# B&R Automation Studio project Foerderband
Automation Studio 4.7.2.98

## Configuration Config1

### Task classes (Cpu.sw)
```
Cyclic#1:
  Program <- Program.prg
Binaries: udbdef, FWRules, TCData, sysconf, Role, User, iomap, ashwd, asiol1, asfw, arconfig, ashwac
Libraries: standard
```

### Hardware
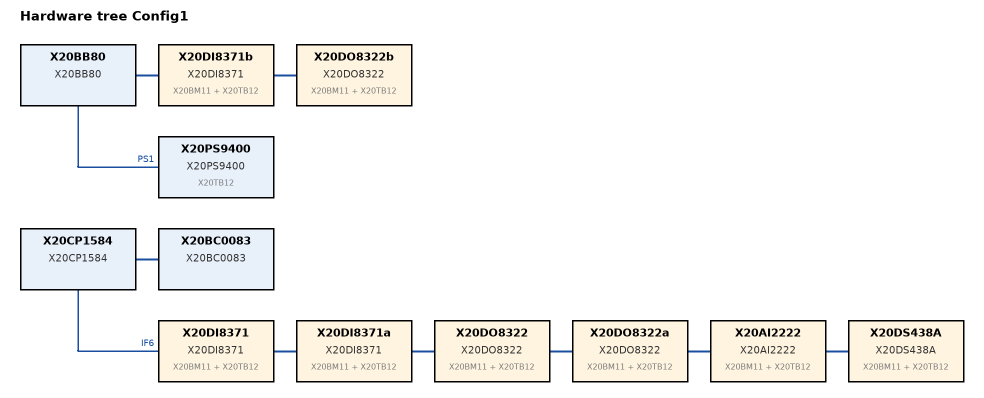
```
X20AI2222 : X20AI2222 v1.0.2.0  [SS1 -> X20TB12d.SS; SL -> X20BM11d.SL1]
X20BB80 : X20BB80 v1.0.2.0
X20BC0083 : X20BC0083 v2.9.0.0  [PLK1 -> X20CP1584.IF3 [Cable Type=PowerlinkCable, Length=10, Version=1.0.0.2]; SL -> X20BB80.SL1]
X20BM11 : X20BM11 v1.0.0.1  [X2X1 -> X20CP1584.IF6]
X20BM11a : X20BM11 v1.0.0.1  [X2X1 -> X20BM11.X2X2]
X20BM11b : X20BM11 v1.0.0.1  [X2X1 -> X20BM11a.X2X2]
X20BM11c : X20BM11 v1.0.0.1  [X2X1 -> X20BM11b.X2X2]
X20BM11d : X20BM11 v1.0.0.1  [X2X1 -> X20BM11c.X2X2]
X20BM11e : X20BM11 v1.0.0.1  [X2X1 -> X20BM11d.X2X2]
X20BM11f : X20BM11 v1.0.0.1  [X2X1 -> X20BB80.IF1]
X20BM11h : X20BM11 v1.0.0.1  [X2X1 -> X20BM11f.X2X2]
X20CP1584 : X20CP1584 v1.6.0.0
  Connector IF2:
    ActivateDevice = 1
    Mode = Manual
    InternetAddress = 10.36.37.4
    SubnetMask = 255.255.255.0
  ConfigurationID = Foerderband_Config1
X20DI8371 : X20DI8371 v1.0.2.0  [SS1 -> X20TB12.SS; SL -> X20BM11.SL1]
X20DI8371a : X20DI8371 v1.0.2.0  [SS1 -> X20TB12a.SS; SL -> X20BM11a.SL1]
X20DI8371b : X20DI8371 v1.0.2.0  [SS1 -> X20TB12f.SS; SL -> X20BM11f.SL1]
X20DO8322 : X20DO8322 v1.1.0.0  [SS1 -> X20TB12b.SS; SL -> X20BM11b.SL1]
X20DO8322a : X20DO8322 v1.1.0.0  [SS1 -> X20TB12c.SS; SL -> X20BM11c.SL1]
X20DO8322b : X20DO8322 v1.1.0.0  [SS1 -> X20TB12i.SS; SL -> X20BM11h.SL1]
X20DS438A : X20DS438A v1.9.1.0  [SS1 -> X20TB12e.SS; SL -> X20BM11e.SL1]
  DtmRef = FBD.BRIOLinkModuleDTM.DTMCore.X20DS438A
  DtmId = 94a64cda-18e3-4e02-9df8-4711ba989a67
  CommDtmId = c69bdead-edba-4600-ad5b-e2199e73abc9
  RequiresDTMBuild = true
  ConfigFile = Communication.dtm
  ConfigModule = asiol1
X20PS9400 : X20PS9400 v1.0.2.4  [SS1 -> X20TB12g.SS; PS -> X20BB80.PS1]
X20TB12 : X20TB12 v1.0.0.0
X20TB12a : X20TB12 v1.0.0.0
X20TB12b : X20TB12 v1.0.0.0
X20TB12c : X20TB12 v1.0.0.0
X20TB12d : X20TB12 v1.0.0.0
X20TB12e : X20TB12 v1.0.0.0
X20TB12f : X20TB12 v1.0.0.0
X20TB12g : X20TB12 v1.0.0.0
X20TB12i : X20TB12 v1.0.0.0
```

### IoMap.iom - X20CP1584/IoMap.iom
```iecst
VAR_CONFIG
	DI_Band_links AT %IX."X20DI8371".DigitalInput01;
	DI_Band_rechts AT %IX."X20DI8371".DigitalInput02;
	DI_Koppel_rechts AT %IX."X20DI8371".DigitalInput03;
	DI_Koppel_links AT %IX."X20DI8371".DigitalInput04;
	DI_Stopper AT %IX."X20DI8371".DigitalInput05;
	DI_NOTAUS AT %IX."X20DI8371".DigitalInput06;
	DI_Drehgeber_1 AT %IX."X20DI8371".DigitalInput07;
	DI_Drehgeber_2  AT %IX."X20DI8371".DigitalInput08;
	DI_Start AT %IX."X20DI8371a".DigitalInput01;
	DI_Stop AT %IX."X20DI8371a".DigitalInput02;
	DI_RESET AT %IX."X20DI8371a".DigitalInput03;
	DI_Wahl AT %IX."X20DI8371a".DigitalInput04;
	DO_Antrieb_rechts AT %QX."X20DO8322".DigitalOutput01;
	DO_Antrieb_links AT %QX."X20DO8322".DigitalOutput02;
	DO_schleichgang AT %QX."X20DO8322".DigitalOutput03;
	DO_Stopper AT %QX."X20DO8322".DigitalOutput04;
	DO_Koppel_links AT %QX."X20DO8322".DigitalOutput05;
	DO_Koppel_rechts AT %QX."X20DO8322".DigitalOutput06;
	DO_gruen AT %QX."X20DO8322a".DigitalOutput01;
	DO_weiss AT %QX."X20DO8322a".DigitalOutput02;
	DO_Q1 AT %QX."X20DO8322a".DigitalOutput03;
	DO_Q2 AT %QX."X20DO8322a".DigitalOutput04;
	AI_Potentiometer_1 AT %IW."X20AI2222".AnalogInput01;
	AI_Potentiometer_2 AT %IW."X20AI2222".AnalogInput02;
END_VAR
```

## Configuration station_1

### Task classes (Cpu.sw)
```
Cyclic#1:
  Foerderban <- Foerderband.prg
  stat_1 <- stat_1.prg
  Foerdeband <- FoerdebandWatch.prg
Binaries: udbdef, FWRules, TCData, sysconf, Role, User, iomap, ashwd, asiol1, asfw, arconfig, ashwac
Libraries: standard
```

### Hardware
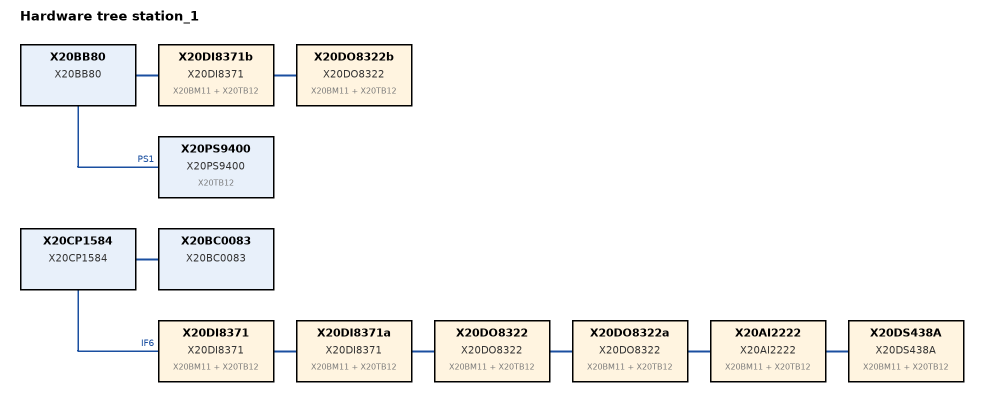
```
X20AI2222 : X20AI2222 v1.0.2.0  [SS1 -> X20TB12d.SS; SL -> X20BM11d.SL1]
X20BB80 : X20BB80 v1.0.2.0
X20BC0083 : X20BC0083 v2.9.0.0  [PLK1 -> X20CP1584.IF3 [Cable Type=PowerlinkCable, Length=10, Version=1.0.0.2]; SL -> X20BB80.SL1]
X20BM11 : X20BM11 v1.0.0.1  [X2X1 -> X20CP1584.IF6]
X20BM11a : X20BM11 v1.0.0.1  [X2X1 -> X20BM11.X2X2]
X20BM11b : X20BM11 v1.0.0.1  [X2X1 -> X20BM11a.X2X2]
X20BM11c : X20BM11 v1.0.0.1  [X2X1 -> X20BM11b.X2X2]
X20BM11d : X20BM11 v1.0.0.1  [X2X1 -> X20BM11c.X2X2]
X20BM11e : X20BM11 v1.0.0.1  [X2X1 -> X20BM11d.X2X2]
X20BM11f : X20BM11 v1.0.0.1  [X2X1 -> X20BB80.IF1]
X20BM11h : X20BM11 v1.0.0.1  [X2X1 -> X20BM11f.X2X2]
X20CP1584 : X20CP1584 v1.6.0.0
  Connector IF2:
    ActivateDevice = 1
    Mode = Manual
    InternetAddress = 10.36.37.1
    SubnetMask = 255.255.255.0
  ConfigurationID = Foerderband_Config1
X20DI8371 : X20DI8371 v1.0.2.0  [SS1 -> X20TB12.SS; SL -> X20BM11.SL1]
X20DI8371a : X20DI8371 v1.0.2.0  [SS1 -> X20TB12a.SS; SL -> X20BM11a.SL1]
X20DI8371b : X20DI8371 v1.0.2.0  [SS1 -> X20TB12f.SS; SL -> X20BM11f.SL1]
X20DO8322 : X20DO8322 v1.1.0.0  [SS1 -> X20TB12b.SS; SL -> X20BM11b.SL1]
X20DO8322a : X20DO8322 v1.1.0.0  [SS1 -> X20TB12c.SS; SL -> X20BM11c.SL1]
X20DO8322b : X20DO8322 v1.1.0.0  [SS1 -> X20TB12i.SS; SL -> X20BM11h.SL1]
X20DS438A : X20DS438A v1.9.1.0  [SS1 -> X20TB12e.SS; SL -> X20BM11e.SL1]
  DtmRef = FBD.BRIOLinkModuleDTM.DTMCore.X20DS438A
  DtmId = 94a64cda-18e3-4e02-9df8-4711ba989a67
  CommDtmId = c69bdead-edba-4600-ad5b-e2199e73abc9
  RequiresDTMBuild = true
  ConfigFile = Communication.dtm
  ConfigModule = asiol1
X20PS9400 : X20PS9400 v1.0.2.4  [SS1 -> X20TB12g.SS; PS -> X20BB80.PS1]
X20TB12 : X20TB12 v1.0.0.0
X20TB12a : X20TB12 v1.0.0.0
X20TB12b : X20TB12 v1.0.0.0
X20TB12c : X20TB12 v1.0.0.0
X20TB12d : X20TB12 v1.0.0.0
X20TB12e : X20TB12 v1.0.0.0
X20TB12f : X20TB12 v1.0.0.0
X20TB12g : X20TB12 v1.0.0.0
X20TB12i : X20TB12 v1.0.0.0
```

### IoMap.iom - X20CP1584/IoMap.iom
```iecst
VAR_CONFIG
	DI_Band_links AT %IX."X20DI8371".DigitalInput01;
	DI_Band_rechts AT %IX."X20DI8371".DigitalInput02;
	DI_Koppel_rechts AT %IX."X20DI8371".DigitalInput03;
	DI_Koppel_links AT %IX."X20DI8371".DigitalInput04;
	DI_Stopper AT %IX."X20DI8371".DigitalInput05;
	DI_NOTAUS AT %IX."X20DI8371".DigitalInput06;
	DI_Drehgeber_1 AT %IX."X20DI8371".DigitalInput07;
	DI_Drehgeber_2 AT %IX."X20DI8371".DigitalInput08;
	DI_Start AT %IX."X20DI8371a".DigitalInput01;
	DI_Stop AT %IX."X20DI8371a".DigitalInput02;
	DI_RESET AT %IX."X20DI8371a".DigitalInput03;
	DI_Wahl AT %IX."X20DI8371a".DigitalInput04;
	DO_Antrieb_rechts AT %QX."X20DO8322".DigitalOutput01;
	DO_Antrieb_links AT %QX."X20DO8322".DigitalOutput02;
	DO_schleichgang AT %QX."X20DO8322".DigitalOutput03;
	DO_Stopper AT %QX."X20DO8322".DigitalOutput04;
	DO_Koppel_links AT %QX."X20DO8322".DigitalOutput05;
	DO_Koppel_rechts AT %QX."X20DO8322".DigitalOutput06;
	DO_gruen AT %QX."X20DO8322a".DigitalOutput01;
	DO_weiss AT %QX."X20DO8322a".DigitalOutput02;
	DO_Q1 AT %QX."X20DO8322a".DigitalOutput03;
	DO_Q2 AT %QX."X20DO8322a".DigitalOutput04;
	AI_Potentiometer_1 AT %IW."X20AI2222".AnalogInput01;
	AI_Potentiometer_2 AT %IW."X20AI2222".AnalogInput02;
	::DI_Ident_1 AT %IX."X20DI8371a".DigitalInput05;
	::DI_Ident_2 AT %IX."X20DI8371a".DigitalInput06;
	::DI_Ident_3 AT %IX."X20DI8371a".DigitalInput07;
	::DI_Ident_4 AT %IX."X20DI8371a".DigitalInput08;
	DI_X_axis_links  AT %IX."X20DI8371b".DigitalInput01;
	DI_X_axis_recht AT %IX."X20DI8371b".DigitalInput02;
	DI_Frontschale_korr  AT %IX."X20DI8371b".DigitalInput03;
	DI_Frontschale_vorh  AT %IX."X20DI8371b".DigitalInput04;
	DI_Z_axis_oben  AT %IX."X20DI8371b".DigitalInput05;
	DI_Z_axis_unten  AT %IX."X20DI8371b".DigitalInput06;
	DI_Deckel_bereits_vorh  AT %IX."X20DI8371b".DigitalInput07;
	DO_X_axis_nach_links  AT %QX."X20DO8322b".DigitalOutput01;
	DO_X_axis_nach_rechts AT %QX."X20DO8322b".DigitalOutput02;
	DO_Z_axis_nach_oben  AT %QX."X20DO8322b".DigitalOutput03;
	DO_Z_axis_nach_unten  AT %QX."X20DO8322b".DigitalOutput04;
	DO_Z_axis_Klemmung  AT %QX."X20DO8322b".DigitalOutput05;
	DO_Bohrer1  AT %QX."X20DO8322b".DigitalOutput06;
	DO_Bohrer2  AT %QX."X20DO8322b".DigitalOutput07;
END_VAR
```

## Configuration station_2

### Task classes (Cpu.sw)
```
Cyclic#1:
  stat_2 <- stat_2.prg
  Foerderban <- Foerderband.prg
  Program <- (binary)
Binaries: udbdef, FWRules, TCData, sysconf, Role, User, iomap, ashwd, asiol1, asfw, arconfig, ashwac
Libraries: standard
```

### Hardware
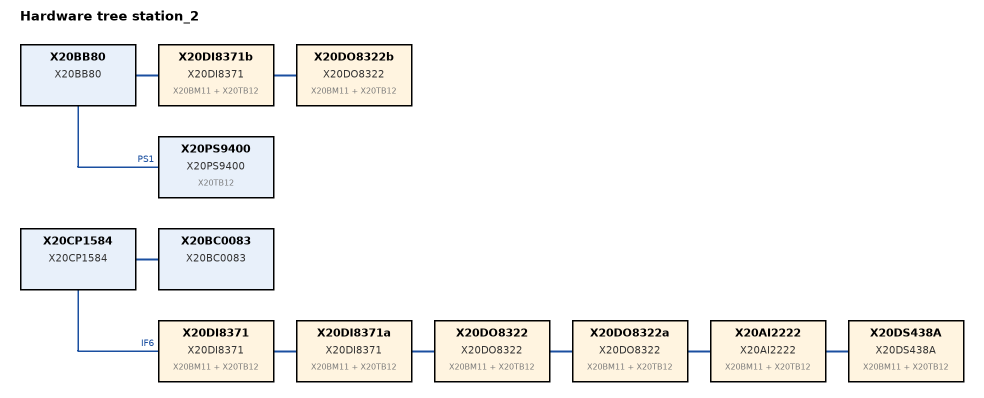
```
X20AI2222 : X20AI2222 v1.0.2.0  [SS1 -> X20TB12d.SS; SL -> X20BM11d.SL1]
X20BB80 : X20BB80 v1.0.2.0
X20BC0083 : X20BC0083 v2.9.0.0  [PLK1 -> X20CP1584.IF3 [Cable Type=PowerlinkCable, Length=10, Version=1.0.0.2]; SL -> X20BB80.SL1]
X20BM11 : X20BM11 v1.0.0.1  [X2X1 -> X20CP1584.IF6]
X20BM11a : X20BM11 v1.0.0.1  [X2X1 -> X20BM11.X2X2]
X20BM11b : X20BM11 v1.0.0.1  [X2X1 -> X20BM11a.X2X2]
X20BM11c : X20BM11 v1.0.0.1  [X2X1 -> X20BM11b.X2X2]
X20BM11d : X20BM11 v1.0.0.1  [X2X1 -> X20BM11c.X2X2]
X20BM11e : X20BM11 v1.0.0.1  [X2X1 -> X20BM11d.X2X2]
X20BM11f : X20BM11 v1.0.0.1  [X2X1 -> X20BB80.IF1]
X20BM11h : X20BM11 v1.0.0.1  [X2X1 -> X20BM11f.X2X2]
X20CP1584 : X20CP1584 v1.6.0.0
  Connector IF2:
    ActivateDevice = 1
    Mode = Manual
    InternetAddress = 10.36.37.2
    SubnetMask = 255.255.255.0
  ConfigurationID = Foerderband_Config1
X20DI8371 : X20DI8371 v1.0.2.0  [SS1 -> X20TB12.SS; SL -> X20BM11.SL1]
X20DI8371a : X20DI8371 v1.0.2.0  [SS1 -> X20TB12a.SS; SL -> X20BM11a.SL1]
X20DI8371b : X20DI8371 v1.0.2.0  [SS1 -> X20TB12f.SS; SL -> X20BM11f.SL1]
X20DO8322 : X20DO8322 v1.1.0.0  [SS1 -> X20TB12b.SS; SL -> X20BM11b.SL1]
X20DO8322a : X20DO8322 v1.1.0.0  [SS1 -> X20TB12c.SS; SL -> X20BM11c.SL1]
X20DO8322b : X20DO8322 v1.1.0.0  [SS1 -> X20TB12i.SS; SL -> X20BM11h.SL1]
X20DS438A : X20DS438A v1.9.1.0  [SS1 -> X20TB12e.SS; SL -> X20BM11e.SL1]
  DtmRef = FBD.BRIOLinkModuleDTM.DTMCore.X20DS438A
  DtmId = 94a64cda-18e3-4e02-9df8-4711ba989a67
  CommDtmId = c69bdead-edba-4600-ad5b-e2199e73abc9
  RequiresDTMBuild = true
  ConfigFile = Communication.dtm
  ConfigModule = asiol1
X20PS9400 : X20PS9400 v1.0.2.4  [SS1 -> X20TB12g.SS; PS -> X20BB80.PS1]
X20TB12 : X20TB12 v1.0.0.0
X20TB12a : X20TB12 v1.0.0.0
X20TB12b : X20TB12 v1.0.0.0
X20TB12c : X20TB12 v1.0.0.0
X20TB12d : X20TB12 v1.0.0.0
X20TB12e : X20TB12 v1.0.0.0
X20TB12f : X20TB12 v1.0.0.0
X20TB12g : X20TB12 v1.0.0.0
X20TB12i : X20TB12 v1.0.0.0
```

### IoMap.iom - X20CP1584/IoMap.iom
```iecst
VAR_CONFIG
	DI_Band_links AT %IX."X20DI8371".DigitalInput01;
	DI_Band_rechts AT %IX."X20DI8371".DigitalInput02;
	DI_Koppel_rechts AT %IX."X20DI8371".DigitalInput03;
	DI_Koppel_links AT %IX."X20DI8371".DigitalInput04;
	DI_Stopper AT %IX."X20DI8371".DigitalInput05;
	DI_NOTAUS AT %IX."X20DI8371".DigitalInput06;
	DI_Drehgeber_1 AT %IX."X20DI8371".DigitalInput07;
	DI_Drehgeber_2 AT %IX."X20DI8371".DigitalInput08;
	DI_Start AT %IX."X20DI8371a".DigitalInput01;
	DI_Stop AT %IX."X20DI8371a".DigitalInput02;
	DI_RESET AT %IX."X20DI8371a".DigitalInput03;
	DI_Wahl AT %IX."X20DI8371a".DigitalInput04;
	DO_Antrieb_rechts AT %QX."X20DO8322".DigitalOutput01;
	DO_Antrieb_links AT %QX."X20DO8322".DigitalOutput02;
	DO_schleichgang AT %QX."X20DO8322".DigitalOutput03;
	DO_Stopper AT %QX."X20DO8322".DigitalOutput04;
	DO_Koppel_links AT %QX."X20DO8322".DigitalOutput05;
	DO_Koppel_rechts AT %QX."X20DO8322".DigitalOutput06;
	DO_gruen AT %QX."X20DO8322a".DigitalOutput01;
	DO_weiss AT %QX."X20DO8322a".DigitalOutput02;
	DO_Q1 AT %QX."X20DO8322a".DigitalOutput03;
	DO_Q2 AT %QX."X20DO8322a".DigitalOutput04;
	AI_Potentiometer_1 AT %IW."X20AI2222".AnalogInput01;
	AI_Potentiometer_2 AT %IW."X20AI2222".AnalogInput02;
	::DI_Ident_1 AT %IX."X20DI8371a".DigitalInput05;
	::DI_Ident_2 AT %IX."X20DI8371a".DigitalInput06;
	::DI_Ident_3 AT %IX."X20DI8371a".DigitalInput07;
	::DI_Ident_4 AT %IX."X20DI8371a".DigitalInput08;
	DI_Hubzylinder_oben  AT %IX."X20DI8371b".DigitalInput01;
	DI_Hubzylinder_unten  AT %IX."X20DI8371b".DigitalInput02;
	DI_untere_Klinge  AT %IX."X20DI8371b".DigitalInput03;
	DI_obere_Klinge  AT %IX."X20DI8371b".DigitalInput04;
	DI_Mag_leer  AT %IX."X20DI8371b".DigitalInput05;
	DI_Palette  AT %IX."X20DI8371b".DigitalInput06;
	DI_Frontschale  AT %IX."X20DI8371b".DigitalInput07;
	DO_Hubzylinder_auf  AT %QX."X20DO8322b".DigitalOutput01;
	DO_Hubzylinder_ab  AT %QX."X20DO8322b".DigitalOutput02;
	DO_Vereinzler_close  AT %QX."X20DO8322b".DigitalOutput03;
	DO_Vereinzler_open  AT %QX."X20DO8322b".DigitalOutput04;
	DO_Zylinderklemmung  AT %QX."X20DO8322b".DigitalOutput05;
END_VAR
```

## Configuration station_3

### Hardware
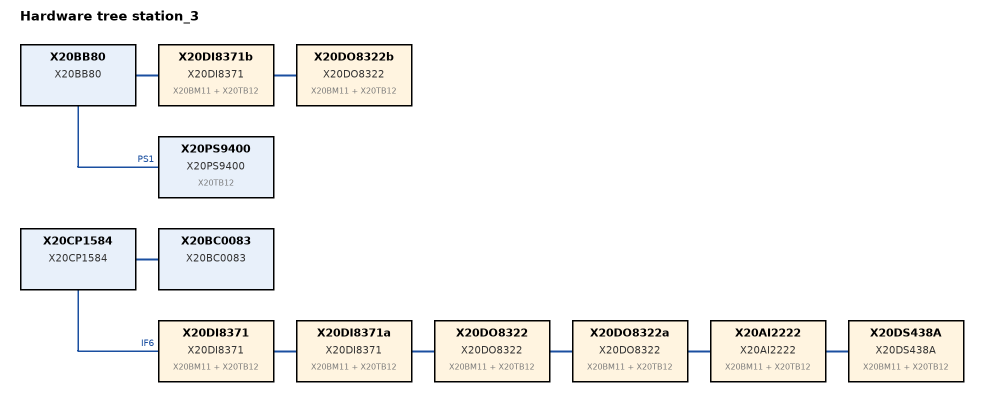
```
X20AI2222 : X20AI2222 v1.0.2.0  [SS1 -> X20TB12d.SS; SL -> X20BM11d.SL1]
X20BB80 : X20BB80 v1.0.2.0
X20BC0083 : X20BC0083 v2.9.0.0  [PLK1 -> X20CP1584.IF3 [Cable Type=PowerlinkCable, Length=10, Version=1.0.0.2]; SL -> X20BB80.SL1]
X20BM11 : X20BM11 v1.0.0.1  [X2X1 -> X20CP1584.IF6]
X20BM11a : X20BM11 v1.0.0.1  [X2X1 -> X20BM11.X2X2]
X20BM11b : X20BM11 v1.0.0.1  [X2X1 -> X20BM11a.X2X2]
X20BM11c : X20BM11 v1.0.0.1  [X2X1 -> X20BM11b.X2X2]
X20BM11d : X20BM11 v1.0.0.1  [X2X1 -> X20BM11c.X2X2]
X20BM11e : X20BM11 v1.0.0.1  [X2X1 -> X20BM11d.X2X2]
X20BM11f : X20BM11 v1.0.0.1  [X2X1 -> X20BB80.IF1]
X20BM11h : X20BM11 v1.0.0.1  [X2X1 -> X20BM11f.X2X2]
X20CP1584 : X20CP1584 v1.6.0.0
  Connector IF2:
    ActivateDevice = 1
    Mode = Manual
    InternetAddress = 10.36.37.3
    SubnetMask = 255.255.255.0
  ConfigurationID = Foerderband_Config1
X20DI8371 : X20DI8371 v1.0.2.0  [SS1 -> X20TB12.SS; SL -> X20BM11.SL1]
X20DI8371a : X20DI8371 v1.0.2.0  [SS1 -> X20TB12a.SS; SL -> X20BM11a.SL1]
X20DI8371b : X20DI8371 v1.0.2.0  [SS1 -> X20TB12f.SS; SL -> X20BM11f.SL1]
X20DO8322 : X20DO8322 v1.1.0.0  [SS1 -> X20TB12b.SS; SL -> X20BM11b.SL1]
X20DO8322a : X20DO8322 v1.1.0.0  [SS1 -> X20TB12c.SS; SL -> X20BM11c.SL1]
X20DO8322b : X20DO8322 v1.1.0.0  [SS1 -> X20TB12i.SS; SL -> X20BM11h.SL1]
X20DS438A : X20DS438A v1.9.1.0  [SS1 -> X20TB12e.SS; SL -> X20BM11e.SL1]
  DtmRef = FBD.BRIOLinkModuleDTM.DTMCore.X20DS438A
  DtmId = 94a64cda-18e3-4e02-9df8-4711ba989a67
  CommDtmId = c69bdead-edba-4600-ad5b-e2199e73abc9
  RequiresDTMBuild = true
  ConfigFile = Communication.dtm
  ConfigModule = asiol1
X20PS9400 : X20PS9400 v1.0.2.4  [SS1 -> X20TB12g.SS; PS -> X20BB80.PS1]
X20TB12 : X20TB12 v1.0.0.0
X20TB12a : X20TB12 v1.0.0.0
X20TB12b : X20TB12 v1.0.0.0
X20TB12c : X20TB12 v1.0.0.0
X20TB12d : X20TB12 v1.0.0.0
X20TB12e : X20TB12 v1.0.0.0
X20TB12f : X20TB12 v1.0.0.0
X20TB12g : X20TB12 v1.0.0.0
X20TB12i : X20TB12 v1.0.0.0
```

### IoMap.iom - X20CP1584/IoMap.iom
```iecst
VAR_CONFIG
	DI_Band_links AT %IX."X20DI8371".DigitalInput01;
	DI_Band_rechts AT %IX."X20DI8371".DigitalInput02;
	DI_Koppel_rechts AT %IX."X20DI8371".DigitalInput03;
	DI_Koppel_links AT %IX."X20DI8371".DigitalInput04;
	DI_Stopper AT %IX."X20DI8371".DigitalInput05;
	DI_NOTAUS AT %IX."X20DI8371".DigitalInput06;
	DI_Drehgeber_1 AT %IX."X20DI8371".DigitalInput07;
	DI_Drehgeber_2 AT %IX."X20DI8371".DigitalInput08;
	DI_Start AT %IX."X20DI8371a".DigitalInput01;
	DI_Stop AT %IX."X20DI8371a".DigitalInput02;
	DI_RESET AT %IX."X20DI8371a".DigitalInput03;
	DI_Wahl AT %IX."X20DI8371a".DigitalInput04;
	DO_Antrieb_rechts AT %QX."X20DO8322".DigitalOutput01;
	DO_Antrieb_links AT %QX."X20DO8322".DigitalOutput02;
	DO_schleichgang AT %QX."X20DO8322".DigitalOutput03;
	DO_Stopper AT %QX."X20DO8322".DigitalOutput04;
	DO_Koppel_links AT %QX."X20DO8322".DigitalOutput05;
	DO_Koppel_rechts AT %QX."X20DO8322".DigitalOutput06;
	DO_gruen AT %QX."X20DO8322a".DigitalOutput01;
	DO_weiss AT %QX."X20DO8322a".DigitalOutput02;
	DO_Q1 AT %QX."X20DO8322a".DigitalOutput03;
	DO_Q2 AT %QX."X20DO8322a".DigitalOutput04;
	AI_Potentiometer_1 AT %IW."X20AI2222".AnalogInput01;
	AI_Potentiometer_2 AT %IW."X20AI2222".AnalogInput02;
	::DI_Ident_1 AT %IX."X20DI8371a".DigitalInput05;
	::DI_Ident_2 AT %IX."X20DI8371a".DigitalInput06;
	::DI_Ident_3 AT %IX."X20DI8371a".DigitalInput07;
	::DI_Ident_4 AT %IX."X20DI8371a".DigitalInput08;
	DI_Hubzylinder_oben_stat3 AT %IX."X20DI8371b".DigitalInput01;
	DI_Hubzylinder_unten_stat3 AT %IX."X20DI8371b".DigitalInput02;
	DI_Frontschale_vorhanden AT %IX."X20DI8371b".DigitalInput03;
	DO_Hubzylinder_auf_stat3 AT %QX."X20DO8322b".DigitalOutput01;
	DO_Hubzylinder_ab_stat3 AT %QX."X20DO8322b".DigitalOutput02;
END_VAR
```

## Configuration station_4

### Task classes (Cpu.sw)
```
Cyclic#1:
  Foerderban <- Foerderband.prg
  stat_4 <- stat_4.prg
Binaries: udbdef, FWRules, TCData, sysconf, Role, User, iomap, ashwd, asiol1, asfw, arconfig, ashwac
Libraries: standard
```

### IoMap.iom - X20CP1584/IoMap.iom
```iecst
VAR_CONFIG
	DI_Band_links AT %IX."X20DI8371".DigitalInput01;
	DI_Band_rechts AT %IX."X20DI8371".DigitalInput02;
	DI_Koppel_rechts AT %IX."X20DI8371".DigitalInput03;
	DI_Koppel_links AT %IX."X20DI8371".DigitalInput04;
	DI_Stopper AT %IX."X20DI8371".DigitalInput05;
	DI_NOTAUS AT %IX."X20DI8371".DigitalInput06;
	DI_Drehgeber_1 AT %IX."X20DI8371".DigitalInput07;
	DI_Drehgeber_2 AT %IX."X20DI8371".DigitalInput08;
	DI_Start AT %IX."X20DI8371a".DigitalInput01;
	DI_Stop AT %IX."X20DI8371a".DigitalInput02;
	DI_RESET AT %IX."X20DI8371a".DigitalInput03;
	DI_Wahl AT %IX."X20DI8371a".DigitalInput04;
	DO_Antrieb_rechts AT %QX."X20DO8322".DigitalOutput01;
	DO_Antrieb_links AT %QX."X20DO8322".DigitalOutput02;
	DO_schleichgang AT %QX."X20DO8322".DigitalOutput03;
	DO_Stopper AT %QX."X20DO8322".DigitalOutput04;
	DO_Koppel_links AT %QX."X20DO8322".DigitalOutput05;
	DO_Koppel_rechts AT %QX."X20DO8322".DigitalOutput06;
	DO_gruen AT %QX."X20DO8322a".DigitalOutput01;
	DO_weiss AT %QX."X20DO8322a".DigitalOutput02;
	DO_Q1 AT %QX."X20DO8322a".DigitalOutput03;
	DO_Q2 AT %QX."X20DO8322a".DigitalOutput04;
	AI_Potentiometer_1 AT %IW."X20AI2222".AnalogInput01;
	AI_Potentiometer_2 AT %IW."X20AI2222".AnalogInput02;
	::DI_Ident_1 AT %IX."X20DI8371a".DigitalInput05;
	::DI_Ident_2 AT %IX."X20DI8371a".DigitalInput06;
	::DI_Ident_3 AT %IX."X20DI8371a".DigitalInput07;
	::DI_Ident_4 AT %IX."X20DI8371a".DigitalInput08;
	DI_Hubzylinder_oben AT %IX."X20DI8371b".DigitalInput01;
	DI_Hubzylinder_unten AT %IX."X20DI8371b".DigitalInput02;
	DI_phi_0 AT %IX."X20DI8371b".DigitalInput03;
	DI_phi_180 AT %IX."X20DI8371b".DigitalInput04;
	DI_Greifer_open AT %IX."X20DI8371b".DigitalInput05;
	DI_Greifer_closed AT %IX."X20DI8371b".DigitalInput06;
	DI_Stau AT %IX."X20DI8371b".DigitalInput07;
	DI_Frontschale AT %IX."X20DI8371b".DigitalInput08;
	DO_Hubzylinder_auf AT %QX."X20DO8322b".DigitalOutput01;
	DO_Hubzylinder_ab AT %QX."X20DO8322b".DigitalOutput02;
	DO_phi_0 AT %QX."X20DO8322b".DigitalOutput03;
	DO_phi_180 AT %QX."X20DO8322b".DigitalOutput04;
	DO_Greifer_open AT %QX."X20DO8322b".DigitalOutput05;
	DO_Greifer_close AT %QX."X20DO8322b".DigitalOutput06;
	DO_Zylinderklemmung AT %QX."X20DO8322b".DigitalOutput07;
END_VAR
```

## Configuration station_5

CPU X20CP1584, AutomationRuntime A4.73, Build 4.1.2, Vc V4.72.0

### Task classes (Cpu.sw)
```
Cyclic#1:
  Foerderban <- Foerderband.prg
  Program <- (binary)
  stat_5 <- stat_5.prg
Binaries: udbdef, FWRules, TCData, sysconf, Role, User, iomap, ashwd, asiol1, asfw, arconfig, ashwac
Libraries: standard
```

### Hardware
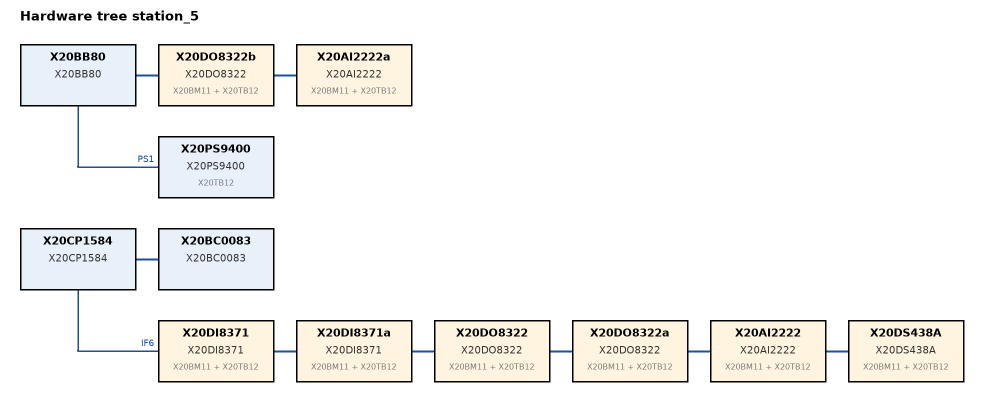
```
X20AI2222 : X20AI2222 v1.0.2.0  [SS1 -> X20TB12d.SS; SL -> X20BM11d.SL1]
X20AI2222a : X20AI2222 v1.0.2.0  [SS1 -> X20TB12h.SS; SL -> X20BM11g.SL1]
X20BB80 : X20BB80 v1.0.2.0
X20BC0083 : X20BC0083 v2.9.0.0  [PLK1 -> X20CP1584.IF3 [Cable Type=PowerlinkCable, Length=10, Version=1.0.0.2]; SL -> X20BB80.SL1]
X20BM11 : X20BM11 v1.0.0.1  [X2X1 -> X20CP1584.IF6]
X20BM11a : X20BM11 v1.0.0.1  [X2X1 -> X20BM11.X2X2]
X20BM11b : X20BM11 v1.0.0.1  [X2X1 -> X20BM11a.X2X2]
X20BM11c : X20BM11 v1.0.0.1  [X2X1 -> X20BM11b.X2X2]
X20BM11d : X20BM11 v1.0.0.1  [X2X1 -> X20BM11c.X2X2]
X20BM11e : X20BM11 v1.0.0.1  [X2X1 -> X20BM11d.X2X2]
X20BM11f : X20BM11 v1.0.0.1  [X2X1 -> X20BB80.IF1]
X20BM11g : X20BM11 v1.0.0.1  [X2X1 -> X20BM11f.X2X2]
X20CP1584 : X20CP1584 v1.6.0.0
  Connector IF2:
    ActivateDevice = 1
    Mode = Manual
    InternetAddress = 10.36.37.5
    SubnetMask = 255.255.255.0
  ConfigurationID = Foerderband_Config1
X20DI8371 : X20DI8371 v1.0.2.0  [SS1 -> X20TB12.SS; SL -> X20BM11.SL1]
X20DI8371a : X20DI8371 v1.0.2.0  [SS1 -> X20TB12a.SS; SL -> X20BM11a.SL1]
X20DO8322 : X20DO8322 v1.1.0.0  [SS1 -> X20TB12b.SS; SL -> X20BM11b.SL1]
X20DO8322a : X20DO8322 v1.1.0.0  [SS1 -> X20TB12c.SS; SL -> X20BM11c.SL1]
X20DO8322b : X20DO8322 v1.1.0.0  [SS1 -> X20TB12f.SS; SL -> X20BM11f.SL1]
X20DS438A : X20DS438A v1.9.1.0  [SS1 -> X20TB12e.SS; SL -> X20BM11e.SL1]
  DtmRef = FBD.BRIOLinkModuleDTM.DTMCore.X20DS438A
  DtmId = 94a64cda-18e3-4e02-9df8-4711ba989a67
  CommDtmId = c69bdead-edba-4600-ad5b-e2199e73abc9
  RequiresDTMBuild = true
  ConfigFile = Communication.dtm
  ConfigModule = asiol1
X20PS9400 : X20PS9400 v1.0.2.4  [SS1 -> X20TB12g.SS; PS -> X20BB80.PS1]
X20TB12 : X20TB12 v1.0.0.0
X20TB12a : X20TB12 v1.0.0.0
X20TB12b : X20TB12 v1.0.0.0
X20TB12c : X20TB12 v1.0.0.0
X20TB12d : X20TB12 v1.0.0.0
X20TB12e : X20TB12 v1.0.0.0
X20TB12f : X20TB12 v1.0.0.0
X20TB12g : X20TB12 v1.0.0.0
X20TB12h : X20TB12 v1.0.0.0
```

### IoMap.iom - X20CP1584/IoMap.iom
```iecst
VAR_CONFIG
	DI_Band_links AT %IX."X20DI8371".DigitalInput01;
	DI_Band_rechts AT %IX."X20DI8371".DigitalInput02;
	DI_Koppel_rechts AT %IX."X20DI8371".DigitalInput03;
	DI_Koppel_links AT %IX."X20DI8371".DigitalInput04;
	DI_Stopper AT %IX."X20DI8371".DigitalInput05;
	DI_NOTAUS AT %IX."X20DI8371".DigitalInput06;
	DI_Drehgeber_1 AT %IX."X20DI8371".DigitalInput07;
	DI_Drehgeber_2 AT %IX."X20DI8371".DigitalInput08;
	DI_Start AT %IX."X20DI8371a".DigitalInput01;
	DI_Stop AT %IX."X20DI8371a".DigitalInput02;
	DI_RESET AT %IX."X20DI8371a".DigitalInput03;
	DI_Wahl AT %IX."X20DI8371a".DigitalInput04;
	DO_Antrieb_rechts AT %QX."X20DO8322".DigitalOutput01;
	DO_Antrieb_links AT %QX."X20DO8322".DigitalOutput02;
	DO_schleichgang AT %QX."X20DO8322".DigitalOutput03;
	DO_Stopper AT %QX."X20DO8322".DigitalOutput04;
	DO_Koppel_links AT %QX."X20DO8322".DigitalOutput05;
	DO_Koppel_rechts AT %QX."X20DO8322".DigitalOutput06;
	DO_gruen AT %QX."X20DO8322a".DigitalOutput01;
	DO_weiss AT %QX."X20DO8322a".DigitalOutput02;
	DO_Q1 AT %QX."X20DO8322a".DigitalOutput03;
	DO_Q2 AT %QX."X20DO8322a".DigitalOutput04;
	AI_Potentiometer_1 AT %IW."X20AI2222".AnalogInput01;
	AI_Potentiometer_2 AT %IW."X20AI2222".AnalogInput02;
	::DI_Ident_1 AT %IX."X20DI8371a".DigitalInput05;
	::DI_Ident_2 AT %IX."X20DI8371a".DigitalInput06;
	::DI_Ident_3 AT %IX."X20DI8371a".DigitalInput07;
	::DI_Ident_4 AT %IX."X20DI8371a".DigitalInput08;
	DO_Heizung AT %QX."X20DO8322b".DigitalOutput01;
	DO_Leistung AT %QX."X20DO8322b".DigitalOutput02;
	AI_Messwandler AT %IW."X20AI2222a".AnalogInput01;
	AI_Messwandler_2 AT %IW."X20AI2222a".AnalogInput02;
END_VAR
```

## Configuration station_6

### Task classes (Cpu.sw)
```
Cyclic#1:
  Foerderban <- Foerderband.prg
  Program <- (binary)
  stat_6 <- stat_6.prg
Binaries: udbdef, FWRules, TCData, sysconf, Role, User, iomap, ashwd, asiol1, asfw, arconfig, ashwac
Libraries: standard
```

### Hardware
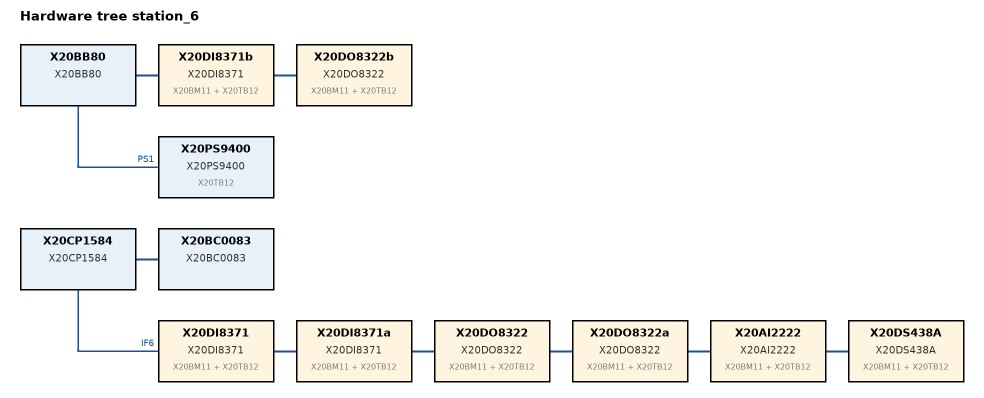
```
X20AI2222 : X20AI2222 v1.0.2.0  [SS1 -> X20TB12d.SS; SL -> X20BM11d.SL1]
X20BB80 : X20BB80 v1.0.2.0
X20BC0083 : X20BC0083 v2.9.0.0  [PLK1 -> X20CP1584.IF3 [Cable Type=PowerlinkCable, Length=10, Version=1.0.0.2]; SL -> X20BB80.SL1]
X20BM11 : X20BM11 v1.0.0.1  [X2X1 -> X20CP1584.IF6]
X20BM11a : X20BM11 v1.0.0.1  [X2X1 -> X20BM11.X2X2]
X20BM11b : X20BM11 v1.0.0.1  [X2X1 -> X20BM11a.X2X2]
X20BM11c : X20BM11 v1.0.0.1  [X2X1 -> X20BM11b.X2X2]
X20BM11d : X20BM11 v1.0.0.1  [X2X1 -> X20BM11c.X2X2]
X20BM11e : X20BM11 v1.0.0.1  [X2X1 -> X20BM11d.X2X2]
X20BM11f : X20BM11 v1.0.0.1  [X2X1 -> X20BB80.IF1]
X20BM11g : X20BM11 v1.0.0.1  [X2X1 -> X20BM11f.X2X2]
X20CP1584 : X20CP1584 v1.6.0.0
  Connector IF2:
    ActivateDevice = 1
    Mode = Manual
    InternetAddress = 10.36.37.6
    SubnetMask = 255.255.255.0
  ConfigurationID = Foerderband_Config1
X20DI8371 : X20DI8371 v1.0.2.0  [SS1 -> X20TB12.SS; SL -> X20BM11.SL1]
X20DI8371a : X20DI8371 v1.0.2.0  [SS1 -> X20TB12a.SS; SL -> X20BM11a.SL1]
X20DI8371b : X20DI8371 v1.0.2.0  [SS1 -> X20TB12g.SS; SL -> X20BM11f.SL1]
X20DO8322 : X20DO8322 v1.1.0.0  [SS1 -> X20TB12b.SS; SL -> X20BM11b.SL1]
X20DO8322a : X20DO8322 v1.1.0.0  [SS1 -> X20TB12c.SS; SL -> X20BM11c.SL1]
X20DO8322b : X20DO8322 v1.1.0.0  [SS1 -> X20TB12h.SS; SL -> X20BM11g.SL1]
X20DS438A : X20DS438A v1.9.1.0  [SS1 -> X20TB12e.SS; SL -> X20BM11e.SL1]
  DtmRef = FBD.BRIOLinkModuleDTM.DTMCore.X20DS438A
  DtmId = 94a64cda-18e3-4e02-9df8-4711ba989a67
  CommDtmId = c69bdead-edba-4600-ad5b-e2199e73abc9
  RequiresDTMBuild = true
  ConfigFile = Communication.dtm
  ConfigModule = asiol1
X20PS9400 : X20PS9400 v1.0.2.4  [SS1 -> X20TB12f.SS; PS -> X20BB80.PS1]
X20TB12 : X20TB12 v1.0.0.0
X20TB12a : X20TB12 v1.0.0.0
X20TB12b : X20TB12 v1.0.0.0
X20TB12c : X20TB12 v1.0.0.0
X20TB12d : X20TB12 v1.0.0.0
X20TB12e : X20TB12 v1.0.0.0
X20TB12f : X20TB12 v1.0.0.0
X20TB12g : X20TB12 v1.0.0.0
X20TB12h : X20TB12 v1.0.0.0
```

### IoMap.iom - X20CP1584/IoMap.iom
```iecst
VAR_CONFIG
	DI_Band_links AT %IX."X20DI8371".DigitalInput01;
	DI_Band_rechts AT %IX."X20DI8371".DigitalInput02;
	DI_Koppel_rechts AT %IX."X20DI8371".DigitalInput03;
	DI_Koppel_links AT %IX."X20DI8371".DigitalInput04;
	DI_Stopper AT %IX."X20DI8371".DigitalInput05;
	DI_NOTAUS AT %IX."X20DI8371".DigitalInput06;
	DI_Drehgeber_1 AT %IX."X20DI8371".DigitalInput07;
	DI_Drehgeber_2 AT %IX."X20DI8371".DigitalInput08;
	DI_Start AT %IX."X20DI8371a".DigitalInput01;
	DI_Stop AT %IX."X20DI8371a".DigitalInput02;
	DI_RESET AT %IX."X20DI8371a".DigitalInput03;
	DI_Wahl AT %IX."X20DI8371a".DigitalInput04;
	DO_Antrieb_rechts AT %QX."X20DO8322".DigitalOutput01;
	DO_Antrieb_links AT %QX."X20DO8322".DigitalOutput02;
	DO_schleichgang AT %QX."X20DO8322".DigitalOutput03;
	DO_Stopper AT %QX."X20DO8322".DigitalOutput04;
	DO_Koppel_links AT %QX."X20DO8322".DigitalOutput05;
	DO_Koppel_rechts AT %QX."X20DO8322".DigitalOutput06;
	DO_gruen AT %QX."X20DO8322a".DigitalOutput01;
	DO_weiss AT %QX."X20DO8322a".DigitalOutput02;
	DO_Q1 AT %QX."X20DO8322a".DigitalOutput03;
	DO_Q2 AT %QX."X20DO8322a".DigitalOutput04;
	AI_Potentiometer_1 AT %IW."X20AI2222".AnalogInput01;
	AI_Potentiometer_2 AT %IW."X20AI2222".AnalogInput02;
	::DI_Ident_1 AT %IX."X20DI8371a".DigitalInput05;
	::DI_Ident_2 AT %IX."X20DI8371a".DigitalInput06;
	::DI_Ident_3 AT %IX."X20DI8371a".DigitalInput07;
	::DI_Ident_4 AT %IX."X20DI8371a".DigitalInput08;
	::stat_6:DI_Kamera_01 AT %IX."X20DI8371b".DigitalInput01;
	::stat_6:DI_Kamera_00 AT %IX."X20DI8371b".DigitalInput02;
	::stat_6:DI_Kamera_02 AT %IX."X20DI8371b".DigitalInput03;
	::stat_6:DO_Kamera_Trigger AT %QX."X20DO8322b".DigitalOutput01;
END_VAR
```

## Logical view

### Global.typ - Global data types
```iecst
TYPE
	error_codes :
		(
		KEIN_ERROR,
		MOTOR_LAEUFT_ZU_LANGE,
		KEINE_DRUCKLUFT,
		ERROR_ANTRIEB
		);
	programm_states :
		(
		EMER_HALT,
		INIT,
		STOP,
		GO_PRE_WORK,
		DETECT,
		WORK,
		GO_AFT_WORK,
		WAIT_TO_LET_GO,
		LET_GO,
		MANUAL,
		ERROR
		);
	koppel_state :
		(
		RTR,
		RTT,
		BUSY
		);
END_TYPE
```

### Global.var - Global variables
```iecst
(*Digital Inputs*)
VAR
	DI_Band_links : BOOL;
	DI_Band_rechts : BOOL;
	DI_Koppel_rechts : BOOL;
	DI_Koppel_links : BOOL;
	DI_Stopper : BOOL;
	DI_NOTAUS : BOOL;
	DI_Drehgeber_1 : BOOL;
	DI_Drehgeber_2 : BOOL;
	DI_Start : BOOL;
	DI_Stop : BOOL;
	DI_RESET : BOOL;
	DI_Wahl : BOOL;
	DI_Ident_1 : BOOL;
	DI_Ident_2 : BOOL;
	DI_Ident_3 : BOOL;
	DI_Ident_4 : BOOL;
END_VAR
(*Digitale Ausgänge*)
VAR
	DO_Antrieb_rechts : BOOL;
	DO_Antrieb_links : BOOL;
	DO_schleichgang : BOOL;
	DO_Stopper : BOOL;
	DO_Koppel_links : BOOL;
	DO_Koppel_rechts : BOOL;
	DO_gruen : BOOL;
	DO_weiss : BOOL;
	DO_Q1 : BOOL;
	DO_Q2 : BOOL;
END_VAR
(*Analoge Eingänge*)
VAR
	AI_Potentiometer_1 : INT;
	AI_Potentiometer_2 : INT;
END_VAR
(*IO_Link*)
VAR
	RFID_Reader : UDINT;
END_VAR
(*Statusvariablen*)
VAR
	manual_work_mode_glob : BOOL;
	auto_mode_glob : USINT;
	work_state : USINT;
	foerderband_state : USINT;
	work_done : BOOL;
	work_now : BOOL;
	set_error_state : BOOL := FALSE;
	error_flag : BOOL := FALSE;
END_VAR
(*Timer*)
VAR CONSTANT
	time_5_s_timer : INT := 5000;
	time_blink_slow : INT := 700;
	time_blink_middle : INT := 375;
	time_blink_fast : INT := 175;
	timer_error_stopper_time : INT := 200;
	timer_error_motor_an_time : INT := 10000;
	heat_timer_time : INT := 12000;
	timer_2s_time : INT := 2000;
END_VAR
VAR
	timer_5s : TON := (0);
	timer_2s : TON;
	timer_error_stopper : TON;
	timer_error : TON;
	timer_blink2 : TON;
	timer_blink : TON;
END_VAR
(*stat_2*)
VAR
	DI_Hubzylinder_oben : BOOL;
	DI_Hubzylinder_unten : BOOL;
	DI_untere_Klinge : BOOL;
	DI_obere_Klinge : BOOL;
	DI_Mag_leer : BOOL;
	DI_Palette : BOOL;
	DI_Frontschale : BOOL;
END_VAR
(*Ausg*)
VAR
	DO_Hubzylinder_auf : BOOL;
	DO_Hubzylinder_ab : BOOL;
	DO_Vereinzler_close : BOOL;
	DO_Vereinzler_open : BOOL;
	DO_Zylinderklemmung : BOOL;
END_VAR
(*stat1*)
VAR
	DI_X_axis_links : BOOL;
	DI_X_axis_recht : BOOL;
	DI_Frontschale_korr : BOOL;
	DI_Frontschale_vorh : BOOL;
	DI_Z_axis_oben : BOOL;
	DI_Deckel_bereits_vorh : BOOL;
	DI_Z_axis_unten : BOOL;
	DO_X_axis_nach_links : BOOL;
	DO_X_axis_nach_rechts : BOOL;
	DO_Z_axis_nach_oben : BOOL;
	DO_Z_axis_nach_unten : BOOL;
	DO_Z_axis_Klemmung : BOOL;
	DO_Bohrer1 : BOOL;
	DO_Bohrer2 : BOOL;
END_VAR
(*stat_3*)
VAR
	DI_Hubzylinder_unten_stat3 : BOOL;
	DI_Hubzylinder_oben_stat3 : BOOL;
	DI_Frontschale_vorhanden : BOOL;
	DO_Hubzylinder_ab_stat3 : BOOL;
	DO_Hubzylinder_auf_stat3 : BOOL;
END_VAR
(*stat_4*)
VAR
	DI_phi_0 : BOOL;
	DI_phi_180 : BOOL;
	DI_Greifer_open : BOOL;
	DI_Greifer_closed : BOOL;
	DI_phi_4 : BOOL;
	DI_Stau : BOOL;
	DI_werkstueck : BOOL;
	DO_phi_0 : BOOL;
	DO_phi_180 : BOOL;
	DO_Greifer_open : BOOL;
	DO_Greifer_close : BOOL;
END_VAR
(*stat_5*)
VAR
	DO_Heizung : BOOL := FALSE;
	DO_Leistung : BOOL := FALSE;
	AI_Messwandler : INT := 0;
	AI_Messwandler_2 : INT := 0;
END_VAR
```

### Program Logical/Foerderband (ANSIC)

#### Variables.var
```iecst
VAR
	timer_blink : TON;
	timer_2s : TON;
	timer_5s : TON;
END_VAR
```

#### Cyclic.c
```c
#define false 0
#define true 1

#include <bur/plctypes.h>
#include <standard.h>

#ifdef _DEFAULT_INCLUDES
#include <AsDefault.h>
#endif

BOOL isWorkMode();
BOOL isAutoMode();
void set_Koppel(enum koppel_state state);
blinkLed(BOOL* led, INT time_to_blink);
blinkLed2(BOOL* led1, BOOL* led2, INT time_to_blink);

void _CYCLIC ProgramCyclic(void)
{
	static enum programm_states state = INIT;
	static enum error_codes error_code = KEIN_ERROR;

	static F_TRIGtyp F_TRIG_01, F_TRIG_autoMode, F_TRIG_rechts;
	static R_TRIGtyp R_TRIG_reset;
	static int auto_mode = false;

	if(!DI_NOTAUS)
		state = EMER_HALT;

	auto_mode = isAutoMode();
	auto_mode_glob = auto_mode;
	work_now = 0;

	switch(state)
	{
		case EMER_HALT:
			DO_Antrieb_rechts = 0;
			DO_Antrieb_links = 0;
			set_Koppel(BUSY);

			if(DI_NOTAUS)
				state = INIT;
			break;

		case INIT:
			DO_gruen = 1;
			DO_Antrieb_rechts = 1;
			DO_Antrieb_links = 0;
			DO_Stopper = 0;
			DO_schleichgang = 0;
			set_Koppel(BUSY);

			timer_2s.IN = 0;
			timer_5s.IN = 1;
			if((DI_Ident_1 || DI_Ident_2 || DI_Ident_3 || DI_Ident_4) && auto_mode)
				state = DETECT;

			if(DI_Band_rechts && auto_mode)
				state = GO_AFT_WORK;

			if(timer_5s.Q && auto_mode)
			{
				timer_5s.IN = 0;
				state = STOP;
			}
			if(!auto_mode)
				state = MANUAL;
			break;

		case STOP:
			DO_Antrieb_rechts = 0;
			DO_Antrieb_links = 0;
			DO_Stopper = 0;
			set_Koppel(RTR);

			timer_2s.IN = 0;

			if(auto_mode && !DI_Koppel_links)
				state = GO_PRE_WORK;
			if(!auto_mode)
			{
				state = MANUAL;
			}
			break;

		case GO_PRE_WORK:
			DO_Antrieb_rechts = 1;
			set_Koppel(RTR);

			timer_2s.IN = 0;

			if((DI_Ident_1 || DI_Ident_2 || DI_Ident_3 || DI_Ident_4) && auto_mode)
				state = DETECT;

			if(!auto_mode)
				state = MANUAL;
			break;

		case DETECT:
			DO_Antrieb_rechts = 1;
			DO_schleichgang = 1;
			set_Koppel(BUSY);

			timer_2s.IN = 1;

			if(timer_2s.Q && auto_mode)
			{
				state = WORK;
				timer_2s.IN = 0;
			}

			if(!auto_mode)
				state = MANUAL;
			break;

		case WORK:
			DO_Antrieb_rechts = 0;
			DO_schleichgang = 0;
			DO_Koppel_links = 0;
			set_Koppel(BUSY);

			timer_2s.IN = 0;
			work_now = 1;

			if(work_done && auto_mode)
				state = GO_AFT_WORK;

			if(!auto_mode)
				state = MANUAL;
			break;

		case GO_AFT_WORK:
			DO_Stopper = 1;
			DO_schleichgang = 0;
			DO_Antrieb_rechts = 1;
			set_Koppel(BUSY);

			timer_2s.IN = 0;

			if(DI_Band_rechts)
				state = WAIT_TO_LET_GO;

			if(!auto_mode)
				state = MANUAL;
			break;

		case WAIT_TO_LET_GO:
			DO_Stopper = 0;
			DO_schleichgang = 0;
			DO_Antrieb_rechts = 0;
			set_Koppel(RTT);

			timer_2s.IN = 0;

			if(!DI_Koppel_rechts) //wait till ÜBERNAHMEBESTÄTIUNGSNACHWEISDOKUMENTENSTEMPEL
				state = LET_GO;

			if(!auto_mode)
				state = MANUAL;
			break;

		case LET_GO: //Let it go, Let it go, can't hold it back anymore :D
			DO_Antrieb_rechts = 1;
			set_Koppel(RTT);

			timer_2s.IN = 0;

			if(auto_mode && !DI_Band_rechts)
				state = STOP;

			if(!auto_mode)
				state = MANUAL;
			break;

		case ERROR:
			DO_Antrieb_links = 0;
			DO_Antrieb_rechts = 0;
			error_flag = true;
			set_Koppel(BUSY);

			timer_2s.IN = 0;
			blinkLed2(&DO_weiss, &DO_gruen, time_blink_fast);

			if(!auto_mode)
				state = MANUAL;
			break;

		case MANUAL:
			set_Koppel(BUSY);
			timer_2s.IN = 0;
			error_flag = 0;

			if (AI_Potentiometer_1 > 16000)
				DO_schleichgang = 0;
			else
				DO_schleichgang = 1;

			if (!manual_work_mode_glob)
			{
				if(DI_Start)
				{
					DO_Antrieb_links = 1;
					DO_Antrieb_rechts = 0;
					DO_weiss = 0;

					if(DO_schleichgang)
						blinkLed(&DO_gruen, time_blink_middle);
					else
						blinkLed(&DO_gruen, time_blink_fast);
				}
				else if(!DO_Antrieb_links && !DI_Stop)
				{
					DO_Antrieb_rechts = 1;
					DO_Antrieb_links = 0;
					DO_gruen = 0;

					if(DO_schleichgang)
						blinkLed(&DO_weiss, time_blink_middle);
					else
						blinkLed(&DO_weiss, time_blink_fast);
				}
				else
				{
					DO_Antrieb_links = 0;
					DO_Antrieb_rechts = 0;

					DO_gruen = 0;
					DO_weiss = 0;
				}

				if(R_TRIG_reset.Q)
				{
					DO_Stopper = !DO_Stopper;
				}
			}
			else
			{
				DO_Antrieb_links = 0;
				DO_Antrieb_rechts = 0;
			}

			if(auto_mode)
			{
				DO_gruen = 0;
				DO_weiss = 0;
				DO_Q1 = 0;
				DO_Q2 = 0;

				state = INIT;
			}
			break;
	}

	DO_Q1 = auto_mode;
	F_TRIG_rechts.CLK = DI_Band_rechts;

	if(DI_Wahl && !auto_mode)
		blinkLed(&DO_gruen, time_blink_slow);

	TON(&timer_2s);
	TON(&timer_5s);
	R_TRIG(&F_TRIG_01);
	R_TRIG_reset.CLK = DI_RESET;
	R_TRIG(&R_TRIG_reset);
	F_TRIG(&F_TRIG_rechts);

	manual_work_mode_glob = isWorkMode();
	DO_Q2 = manual_work_mode_glob;

	foerderband_state = state;

	if(set_error_state)
		state = ERROR;
}

BOOL isWorkMode()
{
	static TON_typ timer;
	static BOOL returnVal = false;

	timer.IN = DI_RESET;
	timer.PT = 2000;

	if(timer.Q)
	{
		returnVal = !returnVal;
		timer.IN = 0;
	}

	if(auto_mode_glob)
		returnVal = false;

	TON(&timer);

	return returnVal;
}

BOOL isAutoMode()
{
	static R_TRIGtyp r_start_but;
	r_start_but.CLK = DI_Start;
	static int auto_mode = false ;

	R_TRIG(&r_start_but);

	if(DI_Wahl)
		if(r_start_but.Q && !error_flag)
			auto_mode = true;
		else ;
	else
	{
		auto_mode = false;
		error_flag = false;
		set_error_state = false;
	}

	if(!DI_Stop)
		auto_mode = false;

	return auto_mode;
}

void set_Koppel(enum koppel_state state)
{
	switch(state)
	{
		case RTR:
			DO_Koppel_links = 1;
			DO_Koppel_rechts = 0;
			break;

		case RTT:
			DO_Koppel_links = !1;
			DO_Koppel_rechts = !0;
			break;

		case BUSY:
			DO_Koppel_links = 0;
			DO_Koppel_rechts = 0;
			break;
	}
}

blinkLed(BOOL* led, INT time_to_blink)
{
	timer_blink.IN = 1;
	timer_blink.PT = time_to_blink;

	TON(&timer_blink);

	if(timer_blink.Q)
	{
		*led = !(*led);
		timer_blink.IN = 0;
		TON(&timer_blink);
	}
}

blinkLed2(BOOL* led_1, BOOL* led_2, INT time_to_blink)
{
	timer_blink2.IN = 1;
	timer_blink2.PT = time_to_blink;

	TON(&timer_blink2);

	if(timer_blink2.Q)
	{
		*led_1 = !(*led_1);
		*led_2 = !(*led_2);
		timer_blink2.IN = 0;
		TON(&timer_blink2);
	}
}
```

#### Init.c
```c
#include <bur/plctypes.h>

#ifdef _DEFAULT_INCLUDES
	#include <AsDefault.h>
#endif

void _INIT ProgramInit(void)
{
	DI_Band_links = 0;
	DI_Band_rechts = 0;
	DI_Koppel_rechts = 0;
	DI_Koppel_links = 0;
	DI_Stopper = 0;
	DI_NOTAUS = 0;
	DI_Drehgeber_1 = 0;
	DI_Drehgeber_2 = 0;
	DI_Start = 0;
	DI_Stop = 0;
	DI_RESET = 0;
	DI_Wahl = 0;
	DI_Ident_1 = DI_Ident_2 = DI_Ident_3 = DI_Ident_4 = 0;

	DO_Antrieb_rechts = 0;
	DO_Antrieb_links = 0;
	DO_schleichgang = 0;
	DO_Stopper = 0;
	DO_Koppel_links = 0;
	DO_Koppel_rechts = 0;
	DO_gruen = 0;
	DO_weiss = 0;
	DO_Q1 = 0;
	DO_Q2 = 0;

	AI_Potentiometer_1 = 0;
	AI_Potentiometer_2 = 0;
	RFID_Reader = 0;

	timer_2s.PT = timer_2s_time;
}
```

### Program Logical/FoerdebandWatch (ANSIC)

#### Cyclic.c
```c
#include <bur/plctypes.h>

#define true 1
#define false 0

#ifdef _DEFAULT_INCLUDES
#include <AsDefault.h>
#endif

void _CYCLIC ProgramCyclic(void)
{
	static enum error_codes error_code = KEIN_ERROR;

	//Stopper ist nicht im gewünschten Zustand / Keine Druckluft vorhanden
	if(DI_Stopper != DO_Stopper)
		timer_error_stopper.IN = 1;
	else
		timer_error_stopper.IN = 0;

	timer_error_stopper.PT = timer_error_stopper_time;
	TON(&timer_error_stopper);

	if(timer_error_stopper.Q)
	{
		timer_error_stopper.IN = 0;
		TON(&timer_error_stopper);

		error_code = KEINE_DRUCKLUFT;
		set_error_state = true;
	}

	//Motor läuft 12 Sekunden (im Automatikmodus)
	if((DO_Antrieb_links || DO_Antrieb_rechts) && auto_mode_glob)
		timer_error.IN = 1;
	else
		timer_error.IN = 0;

	timer_error.PT = timer_error_motor_an_time;
	TON(&timer_error);

	if(timer_error.Q)
	{
		timer_error.IN = 0;
		TON(&timer_error);

		error_code = MOTOR_LAEUFT_ZU_LANGE;
		set_error_state = true;
	}
}
```

#### Init.c
```c
#include <bur/plctypes.h>

#ifdef _DEFAULT_INCLUDES
	#include <AsDefault.h>
#endif

void _INIT ProgramInit(void)
{
}
```

### Program Logical/stat_1 (ANSIC)

#### Types.typ
```iecst
TYPE
	linearStates :
		(
		LINKS,
		RECHTS
		);
	hubzylinderstates :
		(
		UP,
		DWN,
		DONT_MOVE
		);
	states :
		(
		WAIT,
		SENKEN,
		BOHREN,
		VERFAHREN,
		HEBEN,
		FERTIG,
		ERROR_STAT1
		);
END_TYPE
```

#### Cyclic.c
```c
#define false 0
#define true 1
#define OR_MANUAL_MODE(bedingung) ((bedingung)&& auto_mode_glob) || (manual_work_mode_glob && stop_trig.Q)

#include <bur/plctypes.h>
#include <standard.h>

#ifdef _DEFAULT_INCLUDES
#include <AsDefault.h>
#endif

void setHubzylinderstate(enum hubzylinderstates  state);
void setLinearAchse(enum linearStates state);
void setBohrer(int on);

void _CYCLIC ProgramCyclic(void)
{
	static enum states state = WAIT, lastState;
	static F_TRIGtyp stop_trig;
	static TON_typ Error_timer;

	stop_trig.CLK = DI_Stop;
	F_TRIG(&stop_trig);

	switch(state)
	{
		case WAIT:
			setHubzylinderstate(UP);
			setLinearAchse(LINKS);
			setBohrer(0);
			work_done = 0;

			if(OR_MANUAL_MODE(work_now))
				state = BOHREN;
			if(DI_Deckel_bereits_vorh)
				state = FERTIG;
			break;

		case SENKEN:
			setHubzylinderstate(DWN);

			if(OR_MANUAL_MODE(DI_Z_axis_unten))
				state = HEBEN;
			break;

		case BOHREN:
			setBohrer(1);
			state = SENKEN;
			break;

		case VERFAHREN:
			setLinearAchse(RECHTS);

			if(OR_MANUAL_MODE(DI_X_axis_links))
				state = BOHREN;
			break;

		case HEBEN:
			setHubzylinderstate(UP);

			if(OR_MANUAL_MODE(DI_Z_axis_oben))
			{
				if(DI_X_axis_recht)
					state = VERFAHREN;
				else state = FERTIG;
			}
			break;

		case FERTIG:
			work_done = true;

			if(OR_MANUAL_MODE(work_now == 0))
				state = WAIT;
			break;

		case ERROR_STAT1:
			setBohrer(0);
			break;
	}

	if((!auto_mode_glob || !work_now) && !manual_work_mode_glob)
		state = WAIT;

	Error_timer.PT = 4000;
	Error_timer.IN = ((state != WAIT) && (state == lastState));
	TON(&Error_timer);

	if(Error_timer.Q)
		state= ERROR_STAT1;
	lastState=state;
	work_state = state;
}

void setHubzylinderstate(enum hubzylinderstates  state)
{
	DO_Z_axis_Klemmung = 1;

	switch(state)
	{
		case UP:
			DO_Z_axis_nach_oben = 1;
			DO_Z_axis_nach_unten = 0;
			break;

		case DWN:
			DO_Z_axis_nach_oben = 0;
			DO_Z_axis_nach_unten = 1;
			break;

		case DONT_MOVE:
			DO_Z_axis_Klemmung = 0;
			break;
	}
}

void setLinearAchse(enum linearStates state)
{
	switch(state)
	{
		case LINKS:
			DO_X_axis_nach_links = 1;
			DO_X_axis_nach_rechts = 0;
			break;

		case RECHTS:
			DO_X_axis_nach_links = 0;
			DO_X_axis_nach_rechts = 1;
			break;
	}
}

void setBohrer(int on)
{
	DO_Bohrer1 = on;
	DO_Bohrer2 = on;
}
```

#### Init.c
```c
#include <bur/plctypes.h>

#ifdef _DEFAULT_INCLUDES
	#include <AsDefault.h>
#endif

void _INIT ProgramInit(void)
{
	DI_Hubzylinder_oben	=0;
	DI_Hubzylinder_unten=0;
	DI_untere_Klinge=0;
	DI_obere_Klinge=0;
	DI_Mag_leer	=0;
	DI_Palette=0;
	DI_Frontschale=0;

	DO_Hubzylinder_auf=0;
	DO_Hubzylinder_ab=0;
	DO_Vereinzler_close=0;
	DO_Vereinzler_open=0;
	DO_Zylinderklemmung=0;

}
```

### Program Logical/stat_2 (ANSIC)

#### Types.typ
```iecst
TYPE
	hubzylinderstates :
		(
		UP,
		DWN,
		DONT_MOVE
		);
	vereinzlerstates :
		(
		OPEN,
		CLOSE
		);
	states :
		(
		WAIT,
		SENKEN,
		FALLEN_LASSEN,
		HEBEN,
		FERTIG,
		ERROR_STAT2
		);
END_TYPE
```

#### Variables.var
```iecst
VAR
	timer_astable : TON;
END_VAR
```

#### Cyclic.c
```c
#define false 0
#define true 1

#include <bur/plctypes.h>

#ifdef _DEFAULT_INCLUDES
#include <AsDefault.h>
#endif

void setHubzylinderstate(enum hubzylinderstates  state);
void setVereinzlerstate(enum vereinzlerstates state);

void _CYCLIC ProgramCyclic(void)
{
	static enum states state = WAIT;

	switch(state)
	{
		case WAIT:
			setHubzylinderstate(UP);
			setVereinzlerstate(CLOSE);
			work_done = 0;

			if(work_now && DI_Palette)
				state = SENKEN;

			if(DI_Frontschale)
				state = HEBEN;
			break;

		case SENKEN:
			setHubzylinderstate(DWN);

			if(DI_Hubzylinder_unten)
				state = FALLEN_LASSEN;
			break;

		case FALLEN_LASSEN:
			setHubzylinderstate(DONT_MOVE);
			setVereinzlerstate(OPEN);

			if(DI_Hubzylinder_unten && DI_obere_Klinge)
				state = HEBEN;
			break;

		case HEBEN:
			setVereinzlerstate(CLOSE);
			setHubzylinderstate(UP);

			if(DI_Hubzylinder_oben)
				state = FERTIG;
			break;

		case FERTIG:
			work_done = true;
			if(work_now == 0)
				state = WAIT;
			break;

		case ERROR:
			break;
	}

	if(!auto_mode_glob || !work_now)
		state = WAIT;
	work_state = state;
}

void setHubzylinderstate(enum hubzylinderstates  state)
{
	switch(state)
	{
		case UP:
			DO_Hubzylinder_auf = 1;
			DO_Hubzylinder_ab = 0;

			DO_Zylinderklemmung = 1;
			break;

		case DWN:
			DO_Hubzylinder_auf = 0;
			DO_Hubzylinder_ab = 1;

			DO_Zylinderklemmung = 1;
			break;

		case DONT_MOVE:
			DO_Zylinderklemmung = 0;
			break;
	}
}

void setVereinzlerstate(enum vereinzlerstates state)
{
	switch(state)
	{
		case OPEN:
			DO_Vereinzler_close = 0;
			DO_Vereinzler_open = 1;
			break;

		case CLOSE:
			DO_Vereinzler_close = 1;
			DO_Vereinzler_open = 0;
			break;
	}
}
```

#### Init.c
```c
#include <bur/plctypes.h>

#ifdef _DEFAULT_INCLUDES
	#include <AsDefault.h>
#endif

void _INIT ProgramInit(void)
{
	timer_astable.PT = 1500;
	timer_astable.IN = 0;
}
```

### Program Logical/stat_3 (ANSIC)

#### Types.typ
```iecst
TYPE
	hubzylinderstates :
		(
		UP,
		DWN,
		DONT_MOVE
		);
	states :
		(
		WAIT,
		SENKEN,
		HALTEN,
		HEBEN,
		FERTIG,
		ERROR_STAT3
		);
	error_codes_stat3 :
		(
		KEIN_ERROR_STAT3,
		KEINE_FRONTSCHALE_STAT3
		);
END_TYPE
```

#### Variables.var
```iecst
VAR
	Timer_Pressen : TON;
END_VAR
VAR CONSTANT
	Time_Pressen : UINT := 300;
END_VAR
VAR
	error_state_indicator : USINT := 0;
END_VAR
```

#### Cyclic.c
```c
#define false 0
#define true 1

#define OR_MANUAL_MODE(bedingung) ((bedingung)&& auto_mode_glob) || (manual_work_mode_glob && stop_trig.Q)

#include <bur/plctypes.h>

#ifdef _DEFAULT_INCLUDES
#include <AsDefault.h>
#endif

void setHubzylinderstate (enum hubzylinderstates state);

void _CYCLIC ProgramCyclic(void)
{
	static enum states state = WAIT;
	static enum error_codes_stat3 error_codes_stat3 = KEIN_ERROR_STAT3;
	static F_TRIGtyp stop_trig;

	stop_trig.CLK = DI_Stop;
	F_TRIG(&stop_trig);

	switch(state)
	{
		case WAIT:	//Auf Arbeitsbefehl (work_now) warten und überprüfen, ob Frontschale vorhanden
			setHubzylinderstate(UP);
			work_done = 0;
			error_codes_stat3 = KEIN_ERROR_STAT3;

			if((work_now && DI_Frontschale_vorhanden && auto_mode_glob) || (manual_work_mode_glob && stop_trig.Q))	//Arbeitsbefehl vorhanden & Werkstück in Ordnung --> Senken
				state = SENKEN;

			// TODO Testen
			if(work_now && !DI_Frontschale_vorhanden)	//Arbeitsbefehl vorhanden & Werkstück nicht in Ordnung --> Error
			{
				error_codes_stat3 = KEINE_FRONTSCHALE_STAT3;
				error_flag = true;
				state = ERROR_STAT3;
			}
			break;

		case SENKEN:	//Hubzylinder senken und halten
			setHubzylinderstate(DWN);

			if((DI_Hubzylinder_unten_stat3 && auto_mode_glob)|| (manual_work_mode_glob && stop_trig.Q))
				state = HALTEN;
			break;

		case HALTEN:	//Hubzylinder nicht bewegen, Timer abwarten, dann Hubzylinder heben
			setHubzylinderstate(DONT_MOVE);
			Timer_Pressen.IN = 1;

			if ((Timer_Pressen.Q&& auto_mode_glob)|| (manual_work_mode_glob && stop_trig.Q))
			{
				Timer_Pressen.IN = 0;
				state = HEBEN;
			}
			break;

		case HEBEN:		//Hubzylinder heben --> Fertig
			setHubzylinderstate(UP);

			if((DI_Hubzylinder_oben_stat3 && auto_mode_glob)|| (manual_work_mode_glob && stop_trig.Q))
				state = FERTIG;
			break;

		case FERTIG:
			work_done = true;

			if(work_now == 0)
				state = WAIT;
			break;

		case ERROR_STAT3:
			set_error_state = true;

			if(error_flag = 0)
				state = WAIT;
			break;
	}

	if((!auto_mode_glob || !work_now) &&(!manual_work_mode_glob))
		state = WAIT;

	work_state = state;
	TON(&Timer_Pressen);

}

void setHubzylinderstate (enum hubzylinderstates state)
{
	switch(state)
	{
		case UP:
			DO_Hubzylinder_auf_stat3 = 1;
			DO_Hubzylinder_ab_stat3 = 0;
			break;

		case DWN:
			DO_Hubzylinder_auf_stat3 = 0;
			DO_Hubzylinder_ab_stat3 = 1;
			break;

		case DONT_MOVE:
			DO_Hubzylinder_auf_stat3 = 0;
			DO_Hubzylinder_ab_stat3 = 0;
			break;
	}
}
```

#### Init.c
```c
#include <bur/plctypes.h>

#ifdef _DEFAULT_INCLUDES
	#include <AsDefault.h>
#endif

void _INIT ProgramInit(void)
{
	Timer_Pressen.PT = Time_Pressen;
}
```

### Program Logical/stat_4 (ANSIC)

#### Types.typ
```iecst
TYPE
	hubzylinderstates :
		(
		UP,
		DWN,
		DONT_MOVE
		);
	drehzylinderstates :
		(
		_0,
		_180
		);
	greiferstate :
		(
		OPEN,
		CLOSE
		);
	states :
		(
		WAIT,
		GREIFEN,
		LOESEN,
		HEBEN,
		DREHEN,
		SENKEN,
		FERTIG,
		ERROR_STAT4
		);
END_TYPE
```

#### Cyclic.c
```c
#define false 0
#define true 1

#define OR_MANUAL_MODE(bedingung) ((bedingung) && auto_mode_glob) || (manual_work_mode_glob && stop_trig.Q)

#include <bur/plctypes.h>

#ifdef _DEFAULT_INCLUDES
#include <AsDefault.h>
#endif

void setHubzylinderstate(enum hubzylinderstates  state);
void setDrehzylinderstate(enum drehzylinderstates state);
void setGreiferstate(enum greiferstate state);

void _CYCLIC ProgramCyclic(void)
{
	static enum states state = WAIT;
	static F_TRIGtyp stop_trig;

	stop_trig.CLK = DI_Stop;
	F_TRIG(&stop_trig);

	switch(state)
	{
		case WAIT:
			setHubzylinderstate(UP);
			setDrehzylinderstate(_0);
			setGreiferstate(OPEN);

			work_done = 0;

			if(OR_MANUAL_MODE(work_now))
				state = SENKEN;

			if(!DI_Frontschale)
				state = FERTIG;
			break;

		case GREIFEN:
			setGreiferstate(CLOSE);

			if(OR_MANUAL_MODE(DI_Greifer_closed))
				state = HEBEN;
			break;

		case HEBEN:
			setHubzylinderstate(UP);

			if(OR_MANUAL_MODE(DI_Hubzylinder_oben && DI_phi_0))
				state = DREHEN;

			if(OR_MANUAL_MODE(DI_Hubzylinder_oben && DI_phi_180))
				state = FERTIG;
			break;

		case DREHEN:
			setDrehzylinderstate(_180);

			if(OR_MANUAL_MODE(DI_phi_180))
				state = SENKEN;
			break;

		case SENKEN:
			setHubzylinderstate(DWN);

			if(OR_MANUAL_MODE(DI_Hubzylinder_unten && DI_phi_0))
				state = GREIFEN;

			if(OR_MANUAL_MODE(DI_Hubzylinder_unten && DI_phi_180))
				state = LOESEN;
			break;

		case LOESEN:
			setGreiferstate(OPEN);

			if(OR_MANUAL_MODE(DI_Greifer_open))
				state = HEBEN;
			break;

		case FERTIG:
			work_done = true;

			if(work_now == 0)
				state = WAIT;
			break;

		case ERROR_STAT4:
			break;
	}

	if(!auto_mode_glob || !work_now)
		state = WAIT;

	work_state = state;

}

void setHubzylinderstate(enum hubzylinderstates  state)
{
	switch(state)
	{
		case UP:
			DO_Hubzylinder_auf = 1;
			DO_Hubzylinder_ab = 0;
			DO_Zylinderklemmung = 1;
			break;

		case DWN:
			DO_Hubzylinder_auf = 0;
			DO_Hubzylinder_ab = 1;
			DO_Zylinderklemmung = 1;
			break;

		case DONT_MOVE:
			DO_Zylinderklemmung = 0;
			break;
	}
}

void setDrehzylinderstate(enum drehzylinderstates state)
{
	switch(state)
	{
		case _0:
			DO_phi_0 = 1;
			DO_phi_180 = 0;
			break;

		case _180:
			DO_phi_0 = 0;
			DO_phi_180 = 1;
			break;
	}
}

void setGreiferstate(enum greiferstate state)
{
	switch(state)
	{
		case OPEN:
			DO_Greifer_open = 1;
			DO_Greifer_close = 0;
			break;

		case CLOSE:
			DO_Greifer_open = 0;
			DO_Greifer_close = 1;
			break;
	}
}
```

### Program Logical/stat_5 (ANSIC)

#### Types.typ
```iecst
TYPE
	states :
		(
		WAIT,
		HEIZEN,
		FERTIG,
		ERROR_STAT5
		);
END_TYPE
```

#### Cyclic.c
```c
#define TARGET_TEMP 9000
#define HYSTERESE 100

#define false 0
#define true 1

#include <bur/plctypes.h>
#include <standard.h>
#ifdef _DEFAULT_INCLUDES
#include <AsDefault.h>
#endif

enum states{WAIT, HEIZEN, FERTIG, ERROR};

void _CYCLIC ProgramCyclic(void)
{
	static enum states state = WAIT;
	static int _ready_to_go=false;
	static TON_typ heat_timer;
	heat_timer.PT=12000;
	heat_timer.IN=_ready_to_go;
	switch(state)
	{
		case WAIT:
			DO_Heizung = 0;
			work_done = 0;
			_ready_to_go = 0;
			if(work_now)
				state=HEIZEN;
			/*if(!DI_Frontschale)
				state = FERTIG;*/
			break;
		case HEIZEN:
			if(AI_Messwandler > TARGET_TEMP + HYSTERESE/2)
				DO_Heizung = 0;
			if(AI_Messwandler < TARGET_TEMP - HYSTERESE/2)
				DO_Heizung = 1;
			if(AI_Messwandler > TARGET_TEMP)
				_ready_to_go = 1;
			if(heat_timer.Q)
				state=FERTIG;
			break;
		case FERTIG:
			work_done = true;
			DO_Heizung = 0;
			_ready_to_go = 0;
			if(work_now == 0)
				state = WAIT;
			break;
		case ERROR:
			break;
	}
	if(!auto_mode_glob || !work_now)
		state = WAIT;
	work_state = state;
	TON(&heat_timer);
}
```

### Program Logical/stat_6 (ANSIC)

#### Types.typ
```iecst
TYPE
	states_stat6 :
		(
		PROCESS_PIC,
		WORK_DONE,
		TAKE_PIC,
		ERROR_STAT6,
		WAIT
		);
	error_codes_stat6 :
		(
		NO_ERROR,
		SHIT_PIC
		);
END_TYPE
```

#### Variables.var
```iecst
VAR
	DI_Kamera_00 : BOOL := FALSE;
	DI_Kamera_01 : BOOL := FALSE;
	DI_Kamera_02 : BOOL := FALSE;
	DO_Kamera_Trigger : BOOL := FALSE;
	new_pic : BOOL := FALSE;
	timer_picture : TON;
END_VAR
VAR CONSTANT
	timer_picture_time : UINT := 100;
END_VAR
VAR
	nice_pic_cnt : USINT := 0;
	shit_pic_cnt : USINT := 0;
END_VAR
```

#### Cyclic.c
```c
#include <bur/plctypes.h>
#define OR_MANUAL_MODE(bedingung) ((( bedingung ) && auto_mode_glob) || (manual_work_mode_glob && F_TRIG_stop.Q))
#ifdef _DEFAULT_INCLUDES
	#include <AsDefault.h>
#endif

#define true 1
#define false 0
#define TRESHOLD 20

int takePicture(void);
void processPicture(void);

void _CYCLIC ProgramCyclic(void)
{
	static enum states_stat6 state_stat6 = WAIT;
	static enum error_codes_stat6 error_code_stat6 = NO_ERROR;

	static R_TRIGtyp R_TRIG_reset;
	static F_TRIGtyp F_TRIG_stop;

	R_TRIG_reset.CLK = DI_RESET;
	R_TRIG(&R_TRIG_reset);
	F_TRIG_stop.CLK = DI_Stop;
	F_TRIG(&F_TRIG_stop);

	switch(state_stat6)
	{
		case WAIT:
			work_done = false;
			shit_pic_cnt = 0;
			nice_pic_cnt = 0;
			new_pic = 0;

			if(work_now)
				state_stat6 = TAKE_PIC;
			break;

		case TAKE_PIC:	//takes a picture, when finished, switches to processing it
			if(takePicture())
				state_stat6 = PROCESS_PIC;
			break;

		case PROCESS_PIC:	//processes the picture and decides whether its satisfactory or not
			processPicture();

			if((shit_pic_cnt < TRESHOLD) || (nice_pic_cnt < TRESHOLD))
				state_stat6 = TAKE_PIC;

			if(shit_pic_cnt >= TRESHOLD)	//if 10 consecutive pictures are bad -> ERROR_STAT6
			{
				state_stat6 = ERROR_STAT6;
				error_code_stat6 = SHIT_PIC;
			}

			else if (nice_pic_cnt >= TRESHOLD)	//if 10 consecutive pictures are good -> WORK_DONE
				state_stat6 = WORK_DONE;
			break;

		case WORK_DONE:
			work_done = true;

			if(!work_now)
				state_stat6 = WAIT;
			break;

		case ERROR_STAT6:
			if(R_TRIG_reset.Q)
				state_stat6 = WAIT;
			break;
	}
}

int takePicture(void)
{
	timer_picture.IN = true;
	timer_picture.PT = timer_picture_time;
	TON(&timer_picture);

	if(timer_picture.Q)
	{
		DO_Kamera_Trigger = !DO_Kamera_Trigger;
		timer_picture.IN = false;
		TON(&timer_picture);
		new_pic = true;

		return true;
	}
	else
		return false;
}

void processPicture(void)
{
	if(new_pic)
	{
		new_pic = false;

		if (DI_Kamera_00 && (!DI_Kamera_02)) //good pic
			nice_pic_cnt++;

		else if ((!DI_Kamera_00) && DI_Kamera_02)	//bad pic
			shit_pic_cnt++;
	}
}
```

### Program Logical/Program

#### Variables.var
```iecst
VAR
	timer_2s : TON;
	timer_5s : TON;
END_VAR
```

#### Cyclic.c
```c
#define CHECK_CONDITION(params) (params) && isAutoMode()
#define true 1
#define false 0

#include <bur/plctypes.h>
#include <standard.h>

#ifdef _DEFAULT_INCLUDES
#include <AsDefault.h>
#endif

enum error_states{NO_ERROR, TIMEOUT_LEG_1, TIMEOUT_LEG_2, DETECTION_ERROR};
enum programm_states{INIT, STOP, GO_PRE_WORK, DETECT, WORK, GO_AFT_WORK, WAIT_TO_LET_GO, LET_GO, ERROR, TEST};

BOOL isAutoMode()
{
	return 1;
}

void _CYCLIC ProgramCyclic(void)
{
	static enum programm_states state=INIT;
	static enum error_states error= NO_ERROR;
	static R_TRIGtyp r_start_but;
	static F_TRIGtyp F_TRIG_01;
	static int auto_mode=false;

	switch(state)
	{
		case INIT:
			DO_Antrieb_rechts = 1;
			DO_Stopper = 0;

			timer_5s.IN = 1;

			//Schritt 1 im Init: Anlage leer fahren um Fehler durch
			//power loss abzufangen
			if(DI_Band_links)
			{
				state = GO_PRE_WORK;
				timer_5s.IN = 0;
			}
	 		if((DI_Ident_1 || DI_Ident_2 || DI_Ident_3 || DI_Ident_4))
			{
				state=WORK;
				timer_5s.IN = 0;
			}
			if(DI_Band_rechts)
			{
				state=GO_AFT_WORK;
				timer_5s.IN = 0;
			}

			//Wenn die Palette nach 5 Sekunden nirgends aufgetaucht
			//ist, wird wohl keine da sein \O.O/ Was weiß ich,
			//eigentlich isses ja wurscht
			if(timer_5s.Q)
			{
				state = STOP;
				timer_5s.IN = 0;
				DO_Stopper = 0;
			}
			break;
		case STOP:
			DO_Antrieb_rechts = 0;
			DO_Stopper = 0;
			if(DI_Band_links && auto_mode)
				state = GO_PRE_WORK;
			break;
		case GO_PRE_WORK:
			DO_Antrieb_rechts = 1;
			timer_5s.IN = 1;
			if((DI_Ident_1 || DI_Ident_2 || DI_Ident_3 || DI_Ident_4) && auto_mode)
				state = DETECT;
			if(timer_5s.Q && auto_mode)
			{
				state = ERROR;
				timer_5s.IN = 0;
			}
			break;
		case DETECT:
			DO_Antrieb_rechts = 1;
			DO_schleichgang = 1;

			timer_5s.IN = 1;
			timer_2s.IN = 1;
			if(timer_2s.Q && auto_mode)
			{
				state = WORK;
				timer_2s.IN = 0;
				timer_5s.IN = 0;
			}
			break;
		case WORK:
			DO_Antrieb_rechts = 0;
			DO_schleichgang = 0;
			//hier kannste mal arbeiten du Spast
			timer_5s.IN = 1;
			if(timer_5s.Q && auto_mode)
			{
				state = GO_AFT_WORK;
				timer_5s.IN = 0;
			}
			break;
		case GO_AFT_WORK:
			DO_Stopper = 1;
			DO_Antrieb_rechts = 1;
			DO_schleichgang = 0;
			if(DI_Band_rechts)
				state = WAIT_TO_LET_GO;
			break;
		case WAIT_TO_LET_GO:
			DO_Stopper = 0;
			DO_Antrieb_rechts = 0;
			DO_schleichgang = 0;
			DO_Koppel_rechts = 1;
			if(DI_Koppel_rechts) //wait till Übernahmebestätigung
				state = STOP; //eigentlich let go, aber mein rechter Platz ist frei, ich wünsche mir jemanden herbei :(
			break;
		case LET_GO: //Let it go, Let it go, can't hold it back anymore :D
				DO_Koppel_rechts = 0;
				DO_Antrieb_rechts = 0;//eigentlich 0 aber testzwecke
				if(!DI_Koppel_rechts && auto_mode)
					state = STOP;
			break;
		case ERROR:
			break;
	}

	r_start_but.CLK = DI_Start;

	if(DI_Wahl)
		if(r_start_but.Q)
			auto_mode=true;
		else ;
	else
			auto_mode=false;

	DO_Q1 = auto_mode;

	TON(&timer_5s);
	TON(&timer_2s);
	F_TRIG(&F_TRIG_01);
	R_TRIG(&r_start_but);
}
```

#### Init.c
```c
#include <bur/plctypes.h>

#ifdef _DEFAULT_INCLUDES
	#include <AsDefault.h>
#endif

void _INIT ProgramInit(void)
{
	DI_Band_links=0;
	DI_Band_rechts=0;
	DI_Koppel_rechts=0;
	DI_Koppel_links=0;
	DI_Stopper=0;
	DI_NOTAUS=0;
	DI_Drehgeber_1=0;
	DI_Drehgeber_2=0;
	DI_Start=0;
	DI_Stop=0;
	DI_RESET=0;
	DI_Wahl=0;
	DI_Ident_1 = DI_Ident_2 = DI_Ident_3 = DI_Ident_4=0;

	DO_Antrieb_rechts=0;
	DO_Antrieb_links=0;
	DO_schleichgang=0;
	DO_Stopper=0;
	DO_Koppel_links=0;
	DO_Koppel_rechts=0;
	DO_gruen=0;
	DO_weiss=0;
	DO_Q1=0;
	DO_Q2=0;

	AI_Potentiometer_1=0;
	AI_Potentiometer_2=0;
	RFID_Reader=0;

	timer_5s.PT = 5000;
	timer_2s.PT = 2000;
}
```

Listed in the project but not available here: Logical/Libraries
